{attribute addProperty BoxType "BK1250-0000-0000"}
{attribute addProperty Id "Term_397_KL1002KL1002_D229A9CA00"}
{attribute addProperty CRC "2759421257"}
{attribute addProperty SizeInBites "0"}
{attribute addProperty SizeInBytes "0"}
TYPE A_0014_BK1250_0000_0000_A4796D49 EXTENDS BK1250_A5F67C82 :
STRUCT
	{attribute addProperty Name "Term_397_KL1002"}
	Term_397_KL1002 : KL1002_D229A9CA;
END_STRUCT
END_TYPE

(* stored: Version 1.2.0.0, ProductVersion 3.1.4024.9
   DUT A_0014_BK1250_0000_0000_A4796D49: Id {e3953a41-e2c6-40be-b012-01052e234d28} *)
